ABB RobotStudio station: IRB120 Writing.rsstn

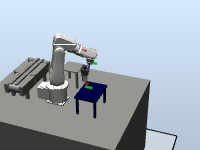
Station Solution4 (saved by RobotStudio 6.8.8148.134)
Controller System1, task T_ROB1: task frame (RAPID world) sits at (85.62, 36.2, 947.96) mm, rotated rx 0 ry 0 rz 180 deg in the station
Controller System1
  mechanical unit ROB_1: IRB120_3_58__01, 6 joints, base frame (0, 0, 0) mm
Layout (positions relative to the parent item):
  - 零件1 [part] at (0, 0, 512.15) mm, rotated rx 90 ry 0 rz 0 deg
  - 写字台 [part] at (-381.08, 197.71, 1142.77) mm, rotated rx 90 ry 0 rz 0 deg
  - 字 [part] at (-241.46, 516.73, 1142.95) mm, rotated rx 90 ry 0 rz 90 deg
  - IRB120_3_58__01 [mechanism, from Robots\IRB120_3_58_G_01.rslib] at (85.62, 36.2, 947.96) mm, rotated rx 0 ry 0 rz 180 deg; joint values [0.5258, 0.1426, 0.3629, -0.5655, 1.4593, 2.276] (rad or m)
  - MyTool [mechanism, from Training Objects\myTool.rslib] at (-205.42, -88.36, 1363.49) mm, rotated rx -180 ry 38 rz -90 deg
  - SmartComponent_1 [smart component]
      signals: DI diTCP
      connections:
        SmartComponent_1.diTCP -> TraceTCP.Enabled
    - TraceTCP [smart component, from Components\TraceTCP.rslib]
        properties: Robot=IRB120_3_58__01
Attachment: MyTool is attached to IRB120_3_58__01 / Link6
Station logic (signal -> signal, property => property):
  System1.doTCP0 -> SmartComponent_1.diTCP
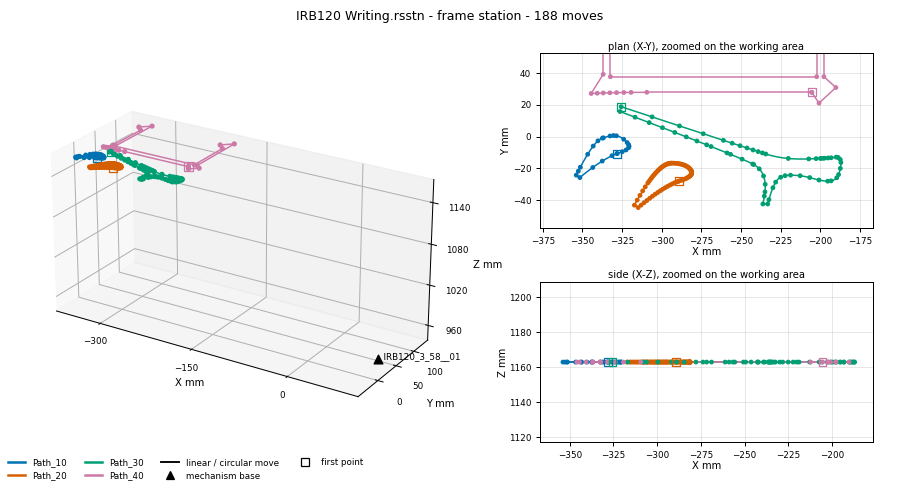
[picture p0: tool path of IRB120 Writing.rsstn in frame station, 188 of 188 moves have a stored position in this frame; points joined in program order, loops and branches not executed]
Targets, tools, work objects and paths stored in the station, written as RAPID:
! task T_ROB1
MODULE Module1
  PERS tooldata MyTool:=[TRUE,[[31.792631019,0,229.638935148],[0.945518576,0,0.325568154,0]],[1,[0,0,1],[1,0,0,0],0,0,0]];
  CONST robtarget Target_10:=[[413.794181769,46.847111716,214.996798109],[0,-0.157825043,0.987467091,0],[0,0,0,0],[9E+09,9E+09,9E+09,9E+09,9E+09,9E+09]];
  CONST robtarget Target_20:=[[415.060758139,47.36953404,214.996798109],[0,-0.157825043,0.987467091,0],[0,0,0,0],[9E+09,9E+09,9E+09,9E+09,9E+09,9E+09]];
  CONST robtarget Target_30:=[[416.985055299,48.218994242,214.996798109],[0,-0.157825043,0.987467091,0],[0,0,0,0],[9E+09,9E+09,9E+09,9E+09,9E+09,9E+09]];
  CONST robtarget Target_40:=[[420.337020954,49.9590146,214.996798109],[0,-0.157825043,0.987467091,0],[0,0,0,0],[9E+09,9E+09,9E+09,9E+09,9E+09,9E+09]];
  CONST robtarget Target_50:=[[423.156723452,51.613418661,214.996798109],[0,-0.157825043,0.987467091,0],[0,0,0,0],[9E+09,9E+09,9E+09,9E+09,9E+09,9E+09]];
  CONST robtarget Target_60:=[[426.087811207,53.506801611,214.996798109],[0,-0.157825043,0.987467091,0],[0,0,0,0],[9E+09,9E+09,9E+09,9E+09,9E+09,9E+09]];
  CONST robtarget Target_70:=[[429.127715578,55.643607322,214.996798109],[0,-0.157825043,0.987467091,0],[0,0,0,0],[9E+09,9E+09,9E+09,9E+09,9E+09,9E+09]];
  CONST robtarget Target_80:=[[433.930399717,59.270989922,214.996798109],[0,-0.157825043,0.987467091,0],[0,0,0,0],[9E+09,9E+09,9E+09,9E+09,9E+09,9E+09]];
  CONST robtarget Target_90:=[[437.267739461,61.991342486,214.996798109],[0,-0.157825043,0.987467091,0],[0,0,0,0],[9E+09,9E+09,9E+09,9E+09,9E+09,9E+09]];
  CONST robtarget Target_100:=[[439.539374076,60.476919409,214.996798109],[0,-0.157825043,0.987467091,0],[0,0,0,0],[9E+09,9E+09,9E+09,9E+09,9E+09,9E+09]];
  CONST robtarget Target_110:=[[438.254894214,57.978091262,214.996798109],[0,-0.157825043,0.987467091,0],[0,0,0,0],[9E+09,9E+09,9E+09,9E+09,9E+09,9E+09]];
  CONST robtarget Target_120:=[[436.959245871,55.484932229,214.996798109],[0,-0.157825043,0.987467091,0],[0,0,0,0],[9E+09,9E+09,9E+09,9E+09,9E+09,9E+09]];
  CONST robtarget Target_130:=[[434.575431769,51.081887357,214.996798109],[0,-0.157825043,0.987467091,0],[0,0,0,0],[9E+09,9E+09,9E+09,9E+09,9E+09,9E+09]];
  CONST robtarget Target_140:=[[432.331842025,47.295829665,214.996798109],[0,-0.157825043,0.987467091,0],[0,0,0,0],[9E+09,9E+09,9E+09,9E+09,9E+09,9E+09]];
  CONST robtarget Target_150:=[[430.790454976,44.888264366,214.996798109],[0,-0.157825043,0.987467091,0],[0,0,0,0],[9E+09,9E+09,9E+09,9E+09,9E+09,9E+09]];
  CONST robtarget Target_160:=[[428.845408894,42.148797629,214.996798109],[0,-0.157825043,0.987467091,0],[0,0,0,0],[9E+09,9E+09,9E+09,9E+09,9E+09,9E+09]];
  CONST robtarget Target_170:=[[427.504490728,40.516553609,214.996798109],[0,-0.157825043,0.987467091,0],[0,0,0,0],[9E+09,9E+09,9E+09,9E+09,9E+09,9E+09]];
  CONST robtarget Target_180:=[[425.856041428,38.831157314,214.996798109],[0,-0.157825043,0.987467091,0],[0,0,0,0],[9E+09,9E+09,9E+09,9E+09,9E+09,9E+09]];
  CONST robtarget Target_190:=[[424.358135134,37.755273557,214.996798109],[0,-0.157825043,0.987467091,0],[0,0,0,0],[9E+09,9E+09,9E+09,9E+09,9E+09,9E+09]];
  CONST robtarget Target_200:=[[423.034428232,37.149604926,214.996798109],[0,-0.157825043,0.987467091,0],[0,0,0,0],[9E+09,9E+09,9E+09,9E+09,9E+09,9E+09]];
  CONST robtarget Target_210:=[[422.419010763,36.934235315,214.996798109],[0,-0.157825043,0.987467091,0],[0,0,0,0],[9E+09,9E+09,9E+09,9E+09,9E+09,9E+09]];
  CONST robtarget Target_220:=[[420.134296252,36.25336216,214.996798109],[0,-0.157825043,0.987467091,0],[0,0,0,0],[9E+09,9E+09,9E+09,9E+09,9E+09,9E+09]];
  CONST robtarget Target_230:=[[418.244052483,35.756988405,214.996798109],[0,-0.157825043,0.987467091,0],[0,0,0,0],[9E+09,9E+09,9E+09,9E+09,9E+09,9E+09]];
  CONST robtarget Target_240:=[[417.383925358,35.601118127,214.996798109],[0,-0.157825043,0.987467091,0],[0,0,0,0],[9E+09,9E+09,9E+09,9E+09,9E+09,9E+09]];
  CONST robtarget Target_250:=[[416.065816384,35.48893864,214.996798109],[0,-0.157825043,0.987467091,0],[0,0,0,0],[9E+09,9E+09,9E+09,9E+09,9E+09,9E+09]];
  CONST robtarget Target_260:=[[415.135685534,35.543807614,214.996798109],[0,-0.157825043,0.987467091,0],[0,0,0,0],[9E+09,9E+09,9E+09,9E+09,9E+09,9E+09]];
  CONST robtarget Target_270:=[[414.214854846,35.65720787,214.996798109],[0,-0.157825043,0.987467091,0],[0,0,0,0],[9E+09,9E+09,9E+09,9E+09,9E+09,9E+09]];
  CONST robtarget Target_280:=[[411.628963846,36.531651758,214.996798109],[0,-0.157825043,0.987467091,0],[0,0,0,0],[9E+09,9E+09,9E+09,9E+09,9E+09,9E+09]];
  CONST robtarget Target_290:=[[409.628567412,37.837626066,214.996798109],[0,-0.157825043,0.987467091,0],[0,0,0,0],[9E+09,9E+09,9E+09,9E+09,9E+09,9E+09]];
  CONST robtarget Target_300:=[[408.575369643,38.75449417,214.996798109],[0,-0.157825043,0.987467091,0],[0,0,0,0],[9E+09,9E+09,9E+09,9E+09,9E+09,9E+09]];
  CONST robtarget Target_310:=[[407.440478174,39.932033456,214.996798109],[0,-0.157825043,0.987467091,0],[0,0,0,0],[9E+09,9E+09,9E+09,9E+09,9E+09,9E+09]];
  CONST robtarget Target_320:=[[406.979277923,40.508970691,214.996798109],[0,-0.157825043,0.987467091,0],[0,0,0,0],[9E+09,9E+09,9E+09,9E+09,9E+09,9E+09]];
  CONST robtarget Target_330:=[[406.528343034,41.21067125,214.996798109],[0,-0.157825043,0.987467091,0],[0,0,0,0],[9E+09,9E+09,9E+09,9E+09,9E+09,9E+09]];
  CONST robtarget Target_340:=[[406.352602418,41.666682817,214.996798109],[0,-0.157825043,0.987467091,0],[0,0,0,0],[9E+09,9E+09,9E+09,9E+09,9E+09,9E+09]];
  CONST robtarget Target_350:=[[406.222066384,42.303842486,214.996798109],[0,-0.157825043,0.987467091,0],[0,0,0,0],[9E+09,9E+09,9E+09,9E+09,9E+09,9E+09]];
  CONST robtarget Target_360:=[[406.291553057,42.730004792,214.996798109],[0,-0.157825043,0.987467091,0],[0,0,0,0],[9E+09,9E+09,9E+09,9E+09,9E+09,9E+09]];
  CONST robtarget Target_370:=[[406.491071898,43.157591418,214.996798109],[0,-0.157825043,0.987467091,0],[0,0,0,0],[9E+09,9E+09,9E+09,9E+09,9E+09,9E+09]];
  CONST robtarget Target_380:=[[407.287771512,44.014579665,214.996798109],[0,-0.157825043,0.987467091,0],[0,0,0,0],[9E+09,9E+09,9E+09,9E+09,9E+09,9E+09]];
  CONST robtarget Target_390:=[[408.129117666,44.575477101,214.996798109],[0,-0.157825043,0.987467091,0],[0,0,0,0],[9E+09,9E+09,9E+09,9E+09,9E+09,9E+09]];
  CONST robtarget Target_400:=[[409.166777923,45.136374537,214.996798109],[0,-0.157825043,0.987467091,0],[0,0,0,0],[9E+09,9E+09,9E+09,9E+09,9E+09,9E+09]];
  CONST robtarget Target_410:=[[410.484886897,45.697271973,214.996798109],[0,-0.157825043,0.987467091,0],[0,0,0,0],[9E+09,9E+09,9E+09,9E+09,9E+09,9E+09]];
  CONST robtarget Target_420:=[[412.027354846,46.286214281,214.996798109],[0,-0.157825043,0.987467091,0],[0,0,0,0],[9E+09,9E+09,9E+09,9E+09,9E+09,9E+09]];
  CONST robtarget Target_430:=[[413.794181769,46.847111716,214.996798109],[0,-0.157825043,0.987467091,0],[0,0,0,0],[9E+09,9E+09,9E+09,9E+09,9E+09,9E+09]];
  CONST robtarget Target_440:=[[375.008124076,64.262977101,214.996798109],[0,0.417358337,0.908741998,0],[0,0,0,0],[9E+09,9E+09,9E+09,9E+09,9E+09,9E+09]];
  CONST robtarget Target_450:=[[376.346419308,64.795791588,214.996798109],[0,0.417358337,0.908741998,0],[0,0,0,0],[9E+09,9E+09,9E+09,9E+09,9E+09,9E+09]];
  CONST robtarget Target_460:=[[377.672386897,65.356727101,214.996798109],[0,0.417358337,0.908741998,0],[0,0,0,0],[9E+09,9E+09,9E+09,9E+09,9E+09,9E+09]];
  CONST robtarget Target_470:=[[379.085741747,66.020298008,214.996798109],[0,0.417358337,0.908741998,0],[0,0,0,0],[9E+09,9E+09,9E+09,9E+09,9E+09,9E+09]];
  CONST robtarget Target_480:=[[380.476874076,66.730925819,214.996798109],[0,0.417358337,0.908741998,0],[0,0,0,0],[9E+09,9E+09,9E+09,9E+09,9E+09,9E+09]];
  CONST robtarget Target_490:=[[381.973257971,67.540696014,214.996798109],[0,0.417358337,0.908741998,0],[0,0,0,0],[9E+09,9E+09,9E+09,9E+09,9E+09,9E+09]];
  CONST robtarget Target_500:=[[383.449630487,68.385573255,214.996798109],[0,0.417358337,0.908741998,0],[0,0,0,0],[9E+09,9E+09,9E+09,9E+09,9E+09,9E+09]];
  CONST robtarget Target_510:=[[385.016861186,69.33557153,214.996798109],[0,0.417358337,0.908741998,0],[0,0,0,0],[9E+09,9E+09,9E+09,9E+09,9E+09,9E+09]];
  CONST robtarget Target_520:=[[386.562611256,70.320669409,214.996798109],[0,0.417358337,0.908741998,0],[0,0,0,0],[9E+09,9E+09,9E+09,9E+09,9E+09,9E+09]];
  CONST robtarget Target_530:=[[388.201363528,71.410852065,214.996798109],[0,0.417358337,0.908741998,0],[0,0,0,0],[9E+09,9E+09,9E+09,9E+09,9E+09,9E+09]];
  CONST robtarget Target_540:=[[389.815816384,72.536214281,214.996798109],[0,0.417358337,0.908741998,0],[0,0,0,0],[9E+09,9E+09,9E+09,9E+09,9E+09,9E+09]];
  CONST robtarget Target_550:=[[391.522124522,73.785045315,214.996798109],[0,0.417358337,0.908741998,0],[0,0,0,0],[9E+09,9E+09,9E+09,9E+09,9E+09,9E+09]];
  CONST robtarget Target_560:=[[393.209245871,75.060252742,214.996798109],[0,0.417358337,0.908741998,0],[0,0,0,0],[9E+09,9E+09,9E+09,9E+09,9E+09,9E+09]];
  CONST robtarget Target_570:=[[394.999763377,76.436392584,214.996798109],[0,0.417358337,0.908741998,0],[0,0,0,0],[9E+09,9E+09,9E+09,9E+09,9E+09,9E+09]];
  CONST robtarget Target_580:=[[396.770944589,77.83669505,214.996798109],[0,0.417358337,0.908741998,0],[0,0,0,0],[9E+09,9E+09,9E+09,9E+09,9E+09,9E+09]];
  CONST robtarget Target_590:=[[398.630982599,79.367934635,214.996798109],[0,0.417358337,0.908741998,0],[0,0,0,0],[9E+09,9E+09,9E+09,9E+09,9E+09,9E+09]];
  CONST robtarget Target_600:=[[400.472867666,80.921630947,214.996798109],[0,0.417358337,0.908741998,0],[0,0,0,0],[9E+09,9E+09,9E+09,9E+09,9E+09,9E+09]];
  CONST robtarget Target_610:=[[402.856681769,79.40720787,214.996798109],[0,0.417358337,0.908741998,0],[0,0,0,0],[9E+09,9E+09,9E+09,9E+09,9E+09,9E+09]];
  CONST robtarget Target_620:=[[401.089854846,76.210092486,214.996798109],[0,0.417358337,0.908741998,0],[0,0,0,0],[9E+09,9E+09,9E+09,9E+09,9E+09,9E+09]];
  CONST robtarget Target_630:=[[399.351072794,73.209291204,214.996798109],[0,0.417358337,0.908741998,0],[0,0,0,0],[9E+09,9E+09,9E+09,9E+09,9E+09,9E+09]];
  CONST robtarget Target_640:=[[397.668380487,70.404804024,214.996798109],[0,0.417358337,0.908741998,0],[0,0,0,0],[9E+09,9E+09,9E+09,9E+09,9E+09,9E+09]];
  CONST robtarget Target_650:=[[396.013733051,67.824675819,214.996798109],[0,0.417358337,0.908741998,0],[0,0,0,0],[9E+09,9E+09,9E+09,9E+09,9E+09,9E+09]];
  CONST robtarget Target_660:=[[394.415175358,65.440861716,214.996798109],[0,0.417358337,0.908741998,0],[0,0,0,0],[9E+09,9E+09,9E+09,9E+09,9E+09,9E+09]];
  CONST robtarget Target_670:=[[393.639289698,64.340440715,214.996798109],[0,0.417358337,0.908741998,0],[0,0,0,0],[9E+09,9E+09,9E+09,9E+09,9E+09,9E+09]];
  CONST robtarget Target_680:=[[392.844662538,63.253361716,214.996798109],[0,0.417358337,0.908741998,0],[0,0,0,0],[9E+09,9E+09,9E+09,9E+09,9E+09,9E+09]];
  CONST robtarget Target_690:=[[392.096719617,62.264585202,214.996798109],[0,0.417358337,0.908741998,0],[0,0,0,0],[9E+09,9E+09,9E+09,9E+09,9E+09,9E+09]];
  CONST robtarget Target_700:=[[391.330239461,61.290220691,214.996798109],[0,0.417358337,0.908741998,0],[0,0,0,0],[9E+09,9E+09,9E+09,9E+09,9E+09,9E+09]];
  CONST robtarget Target_710:=[[390.596978307,60.39852615,214.996798109],[0,0.417358337,0.908741998,0],[0,0,0,0],[9E+09,9E+09,9E+09,9E+09,9E+09,9E+09]];
  CONST robtarget Target_720:=[[389.843861256,59.523393768,214.996798109],[0,0.417358337,0.908741998,0],[0,0,0,0],[9E+09,9E+09,9E+09,9E+09,9E+09,9E+09]];
  CONST robtarget Target_730:=[[389.139301128,58.742195279,214.996798109],[0,0.417358337,0.908741998,0],[0,0,0,0],[9E+09,9E+09,9E+09,9E+09,9E+09,9E+09]];
  CONST robtarget Target_740:=[[388.413572794,57.980925819,214.996798109],[0,0.417358337,0.908741998,0],[0,0,0,0],[9E+09,9E+09,9E+09,9E+09,9E+09,9E+09]];
  CONST robtarget Target_750:=[[387.721616611,57.298552386,214.996798109],[0,0.417358337,0.908741998,0],[0,0,0,0],[9E+09,9E+09,9E+09,9E+09,9E+09,9E+09]];
  CONST robtarget Target_760:=[[387.011329205,56.634771973,214.996798109],[0,0.417358337,0.908741998,0],[0,0,0,0],[9E+09,9E+09,9E+09,9E+09,9E+09,9E+09]];
  CONST robtarget Target_770:=[[386.349253035,56.04656752,214.996798109],[0,0.417358337,0.908741998,0],[0,0,0,0],[9E+09,9E+09,9E+09,9E+09,9E+09,9E+09]];
  CONST robtarget Target_780:=[[385.665175358,55.484932229,214.996798109],[0,0.417358337,0.908741998,0],[0,0,0,0],[9E+09,9E+09,9E+09,9E+09,9E+09,9E+09]];
  CONST robtarget Target_790:=[[385.017465851,55.006494103,214.996798109],[0,0.417358337,0.908741998,0],[0,0,0,0],[9E+09,9E+09,9E+09,9E+09,9E+09,9E+09]];
  CONST robtarget Target_800:=[[384.347066384,54.55945146,214.996798109],[0,0.417358337,0.908741998,0],[0,0,0,0],[9E+09,9E+09,9E+09,9E+09,9E+09,9E+09]];
  CONST robtarget Target_810:=[[383.712063268,54.176492085,214.996798109],[0,0.417358337,0.908741998,0],[0,0,0,0],[9E+09,9E+09,9E+09,9E+09,9E+09,9E+09]];
  CONST robtarget Target_820:=[[383.057002281,53.830284793,214.996798109],[0,0.417358337,0.908741998,0],[0,0,0,0],[9E+09,9E+09,9E+09,9E+09,9E+09,9E+09]];
  CONST robtarget Target_830:=[[382.448312966,53.558411366,214.996798109],[0,0.417358337,0.908741998,0],[0,0,0,0],[9E+09,9E+09,9E+09,9E+09,9E+09,9E+09]];
  CONST robtarget Target_840:=[[381.823027923,53.325477101,214.996798109],[0,0.417358337,0.908741998,0],[0,0,0,0],[9E+09,9E+09,9E+09,9E+09,9E+09,9E+09]];
  CONST robtarget Target_850:=[[381.239521236,53.148696158,214.996798109],[0,0.417358337,0.908741998,0],[0,0,0,0],[9E+09,9E+09,9E+09,9E+09,9E+09,9E+09]];
  CONST robtarget Target_860:=[[380.645143307,53.016983511,214.996798109],[0,0.417358337,0.908741998,0],[0,0,0,0],[9E+09,9E+09,9E+09,9E+09,9E+09,9E+09]];
  CONST robtarget Target_870:=[[380.072473159,52.941341422,214.996798109],[0,0.417358337,0.908741998,0],[0,0,0,0],[9E+09,9E+09,9E+09,9E+09,9E+09,9E+09]];
  CONST robtarget Target_880:=[[379.495303564,52.904804024,214.996798109],[0,0.417358337,0.908741998,0],[0,0,0,0],[9E+09,9E+09,9E+09,9E+09,9E+09,9E+09]];
  CONST robtarget Target_890:=[[378.415082007,52.904711962,214.996798109],[0,0.417358337,0.908741998,0],[0,0,0,0],[9E+09,9E+09,9E+09,9E+09,9E+09,9E+09]];
  CONST robtarget Target_900:=[[377.335848435,52.960893768,214.996798109],[0,0.417358337,0.908741998,0],[0,0,0,0],[9E+09,9E+09,9E+09,9E+09,9E+09,9E+09]];
  CONST robtarget Target_910:=[[376.338043667,53.040496731,214.996798109],[0,0.417358337,0.908741998,0],[0,0,0,0],[9E+09,9E+09,9E+09,9E+09,9E+09,9E+09]];
  CONST robtarget Target_920:=[[375.344662538,53.15720787,214.996798109],[0,0.417358337,0.908741998,0],[0,0,0,0],[9E+09,9E+09,9E+09,9E+09,9E+09,9E+09]];
  CONST robtarget Target_930:=[[374.457782164,53.305987403,214.996798109],[0,0.417358337,0.908741998,0],[0,0,0,0],[9E+09,9E+09,9E+09,9E+09,9E+09,9E+09]];
  CONST robtarget Target_940:=[[373.577835615,53.493746332,214.996798109],[0,0.417358337,0.908741998,0],[0,0,0,0],[9E+09,9E+09,9E+09,9E+09,9E+09,9E+09]];
  CONST robtarget Target_950:=[[372.773048016,53.698879505,214.996798109],[0,0.417358337,0.908741998,0],[0,0,0,0],[9E+09,9E+09,9E+09,9E+09,9E+09,9E+09]];
  CONST robtarget Target_960:=[[371.979277923,53.942464281,214.996798109],[0,0.417358337,0.908741998,0],[0,0,0,0],[9E+09,9E+09,9E+09,9E+09,9E+09,9E+09]];
  CONST robtarget Target_970:=[[371.254081393,54.212783325,214.996798109],[0,0.417358337,0.908741998,0],[0,0,0,0],[9E+09,9E+09,9E+09,9E+09,9E+09,9E+09]];
  CONST robtarget Target_980:=[[370.548989461,54.531406588,214.996798109],[0,0.417358337,0.908741998,0],[0,0,0,0],[9E+09,9E+09,9E+09,9E+09,9E+09,9E+09]];
  CONST robtarget Target_990:=[[369.919037638,54.873733121,214.996798109],[0,0.417358337,0.908741998,0],[0,0,0,0],[9E+09,9E+09,9E+09,9E+09,9E+09,9E+09]];
  CONST robtarget Target_1000:=[[369.315015102,55.260573255,214.996798109],[0,0.417358337,0.908741998,0],[0,0,0,0],[9E+09,9E+09,9E+09,9E+09,9E+09,9E+09]];
  CONST robtarget Target_1010:=[[368.779066824,55.660499694,214.996798109],[0,0.417358337,0.908741998,0],[0,0,0,0],[9E+09,9E+09,9E+09,9E+09,9E+09,9E+09]];
  CONST robtarget Target_1020:=[[368.277354846,56.101919409,214.996798109],[0,0.417358337,0.908741998,0],[0,0,0,0],[9E+09,9E+09,9E+09,9E+09,9E+09,9E+09]];
  CONST robtarget Target_1030:=[[367.832868118,56.571926989,214.996798109],[0,0.417358337,0.908741998,0],[0,0,0,0],[9E+09,9E+09,9E+09,9E+09,9E+09,9E+09]];
  CONST robtarget Target_1040:=[[367.436008692,57.083489922,214.996798109],[0,0.417358337,0.908741998,0],[0,0,0,0],[9E+09,9E+09,9E+09,9E+09,9E+09,9E+09]];
  CONST robtarget Target_1050:=[[367.134505638,57.569713902,214.996798109],[0,0.417358337,0.908741998,0],[0,0,0,0],[9E+09,9E+09,9E+09,9E+09,9E+09,9E+09]];
  CONST robtarget Target_1060:=[[367.008335929,57.826391072,214.996798109],[0,0.417358337,0.908741998,0],[0,0,0,0],[9E+09,9E+09,9E+09,9E+09,9E+09,9E+09]];
  CONST robtarget Target_1070:=[[366.903156128,58.093105306,214.996798109],[0,0.417358337,0.908741998,0],[0,0,0,0],[9E+09,9E+09,9E+09,9E+09,9E+09,9E+09]];
  CONST robtarget Target_1080:=[[366.831717767,58.332956921,214.996798109],[0,0.417358337,0.908741998,0],[0,0,0,0],[9E+09,9E+09,9E+09,9E+09,9E+09,9E+09]];
  CONST robtarget Target_1090:=[[366.782207519,58.578278493,214.996798109],[0,0.417358337,0.908741998,0],[0,0,0,0],[9E+09,9E+09,9E+09,9E+09,9E+09,9E+09]];
  CONST robtarget Target_1100:=[[366.758115486,58.8264061,214.996798109],[0,0.417358337,0.908741998,0],[0,0,0,0],[9E+09,9E+09,9E+09,9E+09,9E+09,9E+09]];
  CONST robtarget Target_1110:=[[366.762931769,59.074675819,214.996798109],[0,0.417358337,0.908741998,0],[0,0,0,0],[9E+09,9E+09,9E+09,9E+09,9E+09,9E+09]];
  CONST robtarget Target_1120:=[[366.799526296,59.323087626,214.996798109],[0,0.417358337,0.908741998,0],[0,0,0,0],[9E+09,9E+09,9E+09,9E+09,9E+09,9E+09]];
  CONST robtarget Target_1130:=[[366.86557166,59.566456761,214.996798109],[0,0.417358337,0.908741998,0],[0,0,0,0],[9E+09,9E+09,9E+09,9E+09,9E+09,9E+09]];
  CONST robtarget Target_1140:=[[366.957420476,59.802316835,214.996798109],[0,0.417358337,0.908741998,0],[0,0,0,0],[9E+09,9E+09,9E+09,9E+09,9E+09,9E+09]];
  CONST robtarget Target_1150:=[[367.071425358,60.02820146,214.996798109],[0,0.417358337,0.908741998,0],[0,0,0,0],[9E+09,9E+09,9E+09,9E+09,9E+09,9E+09]];
  CONST robtarget Target_1160:=[[367.231695097,60.282194269,214.996798109],[0,0.417358337,0.908741998,0],[0,0,0,0],[9E+09,9E+09,9E+09,9E+09,9E+09,9E+09]];
  CONST robtarget Target_1170:=[[367.414118042,60.520052905,214.996798109],[0,0.417358337,0.908741998,0],[0,0,0,0],[9E+09,9E+09,9E+09,9E+09,9E+09,9E+09]];
  CONST robtarget Target_1180:=[[367.828636897,60.953682229,214.996798109],[0,0.417358337,0.908741998,0],[0,0,0,0],[9E+09,9E+09,9E+09,9E+09,9E+09,9E+09]];
  CONST robtarget Target_1190:=[[368.383395251,61.415334756,214.996798109],[0,0.417358337,0.908741998,0],[0,0,0,0],[9E+09,9E+09,9E+09,9E+09,9E+09,9E+09]];
  CONST robtarget Target_1200:=[[368.97847664,61.823073255,214.996798109],[0,0.417358337,0.908741998,0],[0,0,0,0],[9E+09,9E+09,9E+09,9E+09,9E+09,9E+09]];
  CONST robtarget Target_1210:=[[369.749959866,62.269156545,214.996798109],[0,0.417358337,0.908741998,0],[0,0,0,0],[9E+09,9E+09,9E+09,9E+09,9E+09,9E+09]];
  CONST robtarget Target_1220:=[[370.548989461,62.664419409,214.996798109],[0,0.417358337,0.908741998,0],[0,0,0,0],[9E+09,9E+09,9E+09,9E+09,9E+09,9E+09]];
  CONST robtarget Target_1230:=[[371.549209209,63.094640164,214.996798109],[0,0.417358337,0.908741998,0],[0,0,0,0],[9E+09,9E+09,9E+09,9E+09,9E+09,9E+09]];
  CONST robtarget Target_1240:=[[372.56822023,63.477720691,214.996798109],[0,0.417358337,0.908741998,0],[0,0,0,0],[9E+09,9E+09,9E+09,9E+09,9E+09,9E+09]];
  CONST robtarget Target_1250:=[[373.783847633,63.883294038,214.996798109],[0,0.417358337,0.908741998,0],[0,0,0,0],[9E+09,9E+09,9E+09,9E+09,9E+09,9E+09]];
  CONST robtarget Target_1260:=[[375.008124076,64.262977101,214.996798109],[0,0.417358337,0.908741998,0],[0,0,0,0],[9E+09,9E+09,9E+09,9E+09,9E+09,9E+09]];
  CONST robtarget Target_1270:=[[411.186008692,17.315861716,214.996798109],[0,0.150905267,0.988548229,0],[0,0,0,0],[9E+09,9E+09,9E+09,9E+09,9E+09,9E+09]];
  CONST robtarget Target_1280:=[[391.694822794,23.738137357,214.996798109],[0,0.150905267,0.988548229,0],[0,0,0,0],[9E+09,9E+09,9E+09,9E+09,9E+09,9E+09]];
  CONST robtarget Target_1290:=[[374.44722664,29.431246332,214.996798109],[0,0.150905267,0.988548229,0],[0,0,0,0],[9E+09,9E+09,9E+09,9E+09,9E+09,9E+09]];
  CONST robtarget Target_1300:=[[359.44322023,34.339098896,214.996798109],[0,0.150905267,0.988548229,0],[0,0,0,0],[9E+09,9E+09,9E+09,9E+09,9E+09,9E+09]];
  CONST robtarget Target_1310:=[[346.738893307,38.517784793,214.996798109],[0,0.150905267,0.988548229,0],[0,0,0,0],[9E+09,9E+09,9E+09,9E+09,9E+09,9E+09]];
  CONST robtarget Target_1320:=[[341.214053564,40.312656588,214.996798109],[0,0.150905267,0.988548229,0],[0,0,0,0],[9E+09,9E+09,9E+09,9E+09,9E+09,9E+09]];
  CONST robtarget Target_1330:=[[336.250111256,41.911214281,214.996798109],[0,0.150905267,0.988548229,0],[0,0,0,0],[9E+09,9E+09,9E+09,9E+09,9E+09,9E+09]];
  CONST robtarget Target_1340:=[[331.875111256,43.341502742,214.996798109],[0,0.150905267,0.988548229,0],[0,0,0,0],[9E+09,9E+09,9E+09,9E+09,9E+09,9E+09]];
  CONST robtarget Target_1350:=[[328.061008692,44.575477101,214.996798109],[0,0.150905267,0.988548229,0],[0,0,0,0],[9E+09,9E+09,9E+09,9E+09,9E+09,9E+09]];
  CONST robtarget Target_1360:=[[324.807803564,45.613137357,214.996798109],[0,0.150905267,0.988548229,0],[0,0,0,0],[9E+09,9E+09,9E+09,9E+09,9E+09,9E+09]];
  CONST robtarget Target_1370:=[[322.115495871,46.454483511,214.996798109],[0,0.150905267,0.988548229,0],[0,0,0,0],[9E+09,9E+09,9E+09,9E+09,9E+09,9E+09]];
  CONST robtarget Target_1380:=[[319.984085615,47.127560434,214.996798109],[0,0.150905267,0.988548229,0],[0,0,0,0],[9E+09,9E+09,9E+09,9E+09,9E+09,9E+09]];
  CONST robtarget Target_1390:=[[313.085047153,48.894387357,214.996798109],[0,0.150905267,0.988548229,0],[0,0,0,0],[9E+09,9E+09,9E+09,9E+09,9E+09,9E+09]];
  CONST robtarget Target_1400:=[[305.818359796,49.950656798,214.996798109],[0,0.150905267,0.988548229,0],[0,0,0,0],[9E+09,9E+09,9E+09,9E+09,9E+09,9E+09]];
  CONST robtarget Target_1410:=[[299.518531514,50.285951425,214.996798109],[0,0.150905267,0.988548229,0],[0,0,0,0],[9E+09,9E+09,9E+09,9E+09,9E+09,9E+09]];
  CONST robtarget Target_1420:=[[292.934639214,50.217640377,214.996798109],[0,0.150905267,0.988548229,0],[0,0,0,0],[9E+09,9E+09,9E+09,9E+09,9E+09,9E+09]];
  CONST robtarget Target_1430:=[[288.293380487,50.044227101,214.996798109],[0,0.150905267,0.988548229,0],[0,0,0,0],[9E+09,9E+09,9E+09,9E+09,9E+09,9E+09]];
  CONST robtarget Target_1440:=[[285.516938179,49.932047614,214.996798109],[0,0.150905267,0.988548229,0],[0,0,0,0],[9E+09,9E+09,9E+09,9E+09,9E+09,9E+09]];
  CONST robtarget Target_1450:=[[284.26848519,49.869507835,214.996798109],[0,0.150905267,0.988548229,0],[0,0,0,0],[9E+09,9E+09,9E+09,9E+09,9E+09,9E+09]];
  CONST robtarget Target_1460:=[[283.020944589,49.791823255,214.996798109],[0,0.150905267,0.988548229,0],[0,0,0,0],[9E+09,9E+09,9E+09,9E+09,9E+09,9E+09]];
  CONST robtarget Target_1470:=[[280.805399717,49.623554024,214.996798109],[0,0.150905267,0.988548229,0],[0,0,0,0],[9E+09,9E+09,9E+09,9E+09,9E+09,9E+09]];
  CONST robtarget Target_1480:=[[278.81421382,49.483329665,214.996798109],[0,0.150905267,0.988548229,0],[0,0,0,0],[9E+09,9E+09,9E+09,9E+09,9E+09,9E+09]];
  CONST robtarget Target_1490:=[[277.10347664,49.315060434,214.996798109],[0,0.150905267,0.988548229,0],[0,0,0,0],[9E+09,9E+09,9E+09,9E+09,9E+09,9E+09]];
  CONST robtarget Target_1500:=[[275.645143307,49.118746332,214.996798109],[0,0.150905267,0.988548229,0],[0,0,0,0],[9E+09,9E+09,9E+09,9E+09,9E+09,9E+09]];
  CONST robtarget Target_1510:=[[274.969747093,49.178976609,214.996798109],[0,0.150905267,0.988548229,0],[0,0,0,0],[9E+09,9E+09,9E+09,9E+09,9E+09,9E+09]];
  CONST robtarget Target_1520:=[[274.327034333,49.343105306,214.996798109],[0,0.150905267,0.988548229,0],[0,0,0,0],[9E+09,9E+09,9E+09,9E+09,9E+09,9E+09]];
  CONST robtarget Target_1530:=[[273.576969861,49.845534873,214.996798109],[0,0.150905267,0.988548229,0],[0,0,0,0],[9E+09,9E+09,9E+09,9E+09,9E+09,9E+09]];
  CONST robtarget Target_1540:=[[273.031415049,50.632272341,214.996798109],[0,0.150905267,0.988548229,0],[0,0,0,0],[9E+09,9E+09,9E+09,9E+09,9E+09,9E+09]];
  CONST robtarget Target_1550:=[[272.726969299,51.657724944,214.996798109],[0,0.150905267,0.988548229,0],[0,0,0,0],[9E+09,9E+09,9E+09,9E+09,9E+09,9E+09]];
  CONST robtarget Target_1560:=[[272.639258943,52.486789663,214.996798109],[0,0.150905267,0.988548229,0],[0,0,0,0],[9E+09,9E+09,9E+09,9E+09,9E+09,9E+09]];
  CONST robtarget Target_1570:=[[272.700431769,54.503361716,214.996798109],[0,0.150905267,0.988548229,0],[0,0,0,0],[9E+09,9E+09,9E+09,9E+09,9E+09,9E+09]];
  CONST robtarget Target_1580:=[[273.008925358,56.214098896,214.996798109],[0,0.150905267,0.988548229,0],[0,0,0,0],[9E+09,9E+09,9E+09,9E+09,9E+09,9E+09]];
  CONST robtarget Target_1590:=[[273.457643307,58.093105306,214.996798109],[0,0.150905267,0.988548229,0],[0,0,0,0],[9E+09,9E+09,9E+09,9E+09,9E+09,9E+09]];
  CONST robtarget Target_1600:=[[274.13072023,60.112336075,214.996798109],[0,0.150905267,0.988548229,0],[0,0,0,0],[9E+09,9E+09,9E+09,9E+09,9E+09,9E+09]];
  CONST robtarget Target_1610:=[[274.559010932,61.062267847,214.996798109],[0,0.150905267,0.988548229,0],[0,0,0,0],[9E+09,9E+09,9E+09,9E+09,9E+09,9E+09]];
  CONST robtarget Target_1620:=[[275.268769542,62.12463988,214.996798109],[0,0.150905267,0.988548229,0],[0,0,0,0],[9E+09,9E+09,9E+09,9E+09,9E+09,9E+09]];
  CONST robtarget Target_1630:=[[276.826598747,63.357179665,214.996798109],[0,0.150905267,0.988548229,0],[0,0,0,0],[9E+09,9E+09,9E+09,9E+09,9E+09,9E+09]];
  CONST robtarget Target_1640:=[[278.829760733,64.072101822,214.996798109],[0,0.150905267,0.988548229,0],[0,0,0,0],[9E+09,9E+09,9E+09,9E+09,9E+09,9E+09]];
  CONST robtarget Target_1650:=[[279.729661692,64.19159225,214.996798109],[0,0.150905267,0.988548229,0],[0,0,0,0],[9E+09,9E+09,9E+09,9E+09,9E+09,9E+09]];
  CONST robtarget Target_1660:=[[280.945624076,64.262977101,214.996798109],[0,0.150905267,0.988548229,0],[0,0,0,0],[9E+09,9E+09,9E+09,9E+09,9E+09,9E+09]];
  CONST robtarget Target_1670:=[[283.732571069,64.043896483,214.996798109],[0,0.150905267,0.988548229,0],[0,0,0,0],[9E+09,9E+09,9E+09,9E+09,9E+09,9E+09]];
  CONST robtarget Target_1680:=[[286.45346803,63.535976952,214.996798109],[0,0.150905267,0.988548229,0],[0,0,0,0],[9E+09,9E+09,9E+09,9E+09,9E+09,9E+09]];
  CONST robtarget Target_1690:=[[288.742098435,62.972912998,214.996798109],[0,0.150905267,0.988548229,0],[0,0,0,0],[9E+09,9E+09,9E+09,9E+09,9E+09,9E+09]];
  CONST robtarget Target_1700:=[[292.303797153,61.991342486,214.996798109],[0,0.150905267,0.988548229,0],[0,0,0,0],[9E+09,9E+09,9E+09,9E+09,9E+09,9E+09]];
  CONST robtarget Target_1710:=[[295.323474875,61.342771747,214.996798109],[0,0.150905267,0.988548229,0],[0,0,0,0],[9E+09,9E+09,9E+09,9E+09,9E+09,9E+09]];
  CONST robtarget Target_1720:=[[298.361489461,60.841502742,214.996798109],[0,0.150905267,0.988548229,0],[0,0,0,0],[9E+09,9E+09,9E+09,9E+09,9E+09,9E+09]];
  CONST robtarget Target_1730:=[[301.381453975,60.587864036,214.996798109],[0,0.150905267,0.988548229,0],[0,0,0,0],[9E+09,9E+09,9E+09,9E+09,9E+09,9E+09]];
  CONST robtarget Target_1740:=[[304.419181769,60.476919409,214.996798109],[0,0.150905267,0.988548229,0],[0,0,0,0],[9E+09,9E+09,9E+09,9E+09,9E+09,9E+09]];
  CONST robtarget Target_1750:=[[305.823944153,60.555611726,214.996798109],[0,0.150905267,0.988548229,0],[0,0,0,0],[9E+09,9E+09,9E+09,9E+09,9E+09,9E+09]];
  CONST robtarget Target_1760:=[[307.839452971,60.804320879,214.996798109],[0,0.150905267,0.988548229,0],[0,0,0,0],[9E+09,9E+09,9E+09,9E+09,9E+09,9E+09]];
  CONST robtarget Target_1770:=[[309.344399588,61.20780969,214.996798109],[0,0.150905267,0.988548229,0],[0,0,0,0],[9E+09,9E+09,9E+09,9E+09,9E+09,9E+09]];
  CONST robtarget Target_1780:=[[310.637356728,61.801774962,214.996798109],[0,0.150905267,0.988548229,0],[0,0,0,0],[9E+09,9E+09,9E+09,9E+09,9E+09,9E+09]];
  CONST robtarget Target_1790:=[[312.391609876,63.105831359,214.996798109],[0,0.150905267,0.988548229,0],[0,0,0,0],[9E+09,9E+09,9E+09,9E+09,9E+09,9E+09]];
  CONST robtarget Target_1800:=[[313.786168948,64.879964281,214.996798109],[0,0.150905267,0.988548229,0],[0,0,0,0],[9E+09,9E+09,9E+09,9E+09,9E+09,9E+09]];
  CONST robtarget Target_1810:=[[314.821293413,66.823617905,214.996798109],[0,0.150905267,0.988548229,0],[0,0,0,0],[9E+09,9E+09,9E+09,9E+09,9E+09,9E+09]];
  CONST robtarget Target_1820:=[[315.519541802,68.424094217,214.996798109],[0,0.150905267,0.988548229,0],[0,0,0,0],[9E+09,9E+09,9E+09,9E+09,9E+09,9E+09]];
  CONST robtarget Target_1830:=[[316.965497265,72.350515519,214.996798109],[0,0.150905267,0.988548229,0],[0,0,0,0],[9E+09,9E+09,9E+09,9E+09,9E+09,9E+09]];
  CONST robtarget Target_1840:=[[318.048989461,75.929643768,214.996798109],[0,0.150905267,0.988548229,0],[0,0,0,0],[9E+09,9E+09,9E+09,9E+09,9E+09,9E+09]];
  CONST robtarget Target_1850:=[[318.806200999,78.649996332,214.996798109],[0,0.150905267,0.988548229,0],[0,0,0,0],[9E+09,9E+09,9E+09,9E+09,9E+09,9E+09]];
  CONST robtarget Target_1860:=[[321.835047153,78.649996332,214.996798109],[0,0.150905267,0.988548229,0],[0,0,0,0],[9E+09,9E+09,9E+09,9E+09,9E+09,9E+09]];
  CONST robtarget Target_1870:=[[321.316970665,76.022937631,214.996798109],[0,0.150905267,0.988548229,0],[0,0,0,0],[9E+09,9E+09,9E+09,9E+09,9E+09,9E+09]];
  CONST robtarget Target_1880:=[[320.931127923,73.673514776,214.996798109],[0,0.150905267,0.988548229,0],[0,0,0,0],[9E+09,9E+09,9E+09,9E+09,9E+09,9E+09]];
  CONST robtarget Target_1890:=[[320.539802408,71.023557328,214.996798109],[0,0.150905267,0.988548229,0],[0,0,0,0],[9E+09,9E+09,9E+09,9E+09,9E+09,9E+09]];
  CONST robtarget Target_1900:=[[320.35022474,68.947563161,214.996798109],[0,0.150905267,0.988548229,0],[0,0,0,0],[9E+09,9E+09,9E+09,9E+09,9E+09,9E+09]];
  CONST robtarget Target_1910:=[[320.389794073,66.260140652,214.996798109],[0,0.150905267,0.988548229,0],[0,0,0,0],[9E+09,9E+09,9E+09,9E+09,9E+09,9E+09]];
  CONST robtarget Target_1920:=[[320.741297153,63.477720691,214.996798109],[0,0.150905267,0.988548229,0],[0,0,0,0],[9E+09,9E+09,9E+09,9E+09,9E+09,9E+09]];
  CONST robtarget Target_1930:=[[321.440572753,60.993804489,214.996798109],[0,0.150905267,0.988548229,0],[0,0,0,0],[9E+09,9E+09,9E+09,9E+09,9E+09,9E+09]];
  CONST robtarget Target_1940:=[[322.479629289,58.791360356,214.996798109],[0,0.150905267,0.988548229,0],[0,0,0,0],[9E+09,9E+09,9E+09,9E+09,9E+09,9E+09]];
  CONST robtarget Target_1950:=[[324.162771512,56.494547614,214.996798109],[0,0.150905267,0.988548229,0],[0,0,0,0],[9E+09,9E+09,9E+09,9E+09,9E+09,9E+09]];
  CONST robtarget Target_1960:=[[325.920129397,54.873411323,214.996798109],[0,0.150905267,0.988548229,0],[0,0,0,0],[9E+09,9E+09,9E+09,9E+09,9E+09,9E+09]];
  CONST robtarget Target_1970:=[[327.691316065,53.736725754,214.996798109],[0,0.150905267,0.988548229,0],[0,0,0,0],[9E+09,9E+09,9E+09,9E+09,9E+09,9E+09]];
  CONST robtarget Target_1980:=[[328.257322794,53.437656588,214.996798109],[0,0.150905267,0.988548229,0],[0,0,0,0],[9E+09,9E+09,9E+09,9E+09,9E+09,9E+09]];
  CONST robtarget Target_1990:=[[331.059639589,52.100628217,214.996798109],[0,0.150905267,0.988548229,0],[0,0,0,0],[9E+09,9E+09,9E+09,9E+09,9E+09,9E+09]];
  CONST robtarget Target_2000:=[[334.988092025,50.380765563,214.996798109],[0,0.150905267,0.988548229,0],[0,0,0,0],[9E+09,9E+09,9E+09,9E+09,9E+09,9E+09]];
  CONST robtarget Target_2010:=[[342.25171382,47.351919409,214.996798109],[0,0.150905267,0.988548229,0],[0,0,0,0],[9E+09,9E+09,9E+09,9E+09,9E+09,9E+09]];
  CONST robtarget Target_2020:=[[344.47889143,46.448622881,214.996798109],[0,0.150905267,0.988548229,0],[0,0,0,0],[9E+09,9E+09,9E+09,9E+09,9E+09,9E+09]];
  CONST robtarget Target_2030:=[[354.533547438,42.425438051,214.996798109],[0,0.150905267,0.988548229,0],[0,0,0,0],[9E+09,9E+09,9E+09,9E+09,9E+09,9E+09]];
  CONST robtarget Target_2040:=[[357.311809974,41.322271973,214.996798109],[0,0.150905267,0.988548229,0],[0,0,0,0],[9E+09,9E+09,9E+09,9E+09,9E+09,9E+09]];
  CONST robtarget Target_2050:=[[363.453636897,38.93845787,214.996798109],[0,0.150905267,0.988548229,0],[0,0,0,0],[9E+09,9E+09,9E+09,9E+09,9E+09,9E+09]];
  CONST robtarget Target_2060:=[[370.156361256,36.330284793,214.996798109],[0,0.150905267,0.988548229,0],[0,0,0,0],[9E+09,9E+09,9E+09,9E+09,9E+09,9E+09]];
  CONST robtarget Target_2070:=[[377.391938179,33.525797614,214.996798109],[0,0.150905267,0.988548229,0],[0,0,0,0],[9E+09,9E+09,9E+09,9E+09,9E+09,9E+09]];
  CONST robtarget Target_2080:=[[385.188412538,30.524996332,214.996798109],[0,0.150905267,0.988548229,0],[0,0,0,0],[9E+09,9E+09,9E+09,9E+09,9E+09,9E+09]];
  CONST robtarget Target_2090:=[[393.545784333,27.327880947,214.996798109],[0,0.150905267,0.988548229,0],[0,0,0,0],[9E+09,9E+09,9E+09,9E+09,9E+09,9E+09]];
  CONST robtarget Target_2100:=[[402.464053564,23.93445146,214.996798109],[0,0.150905267,0.988548229,0],[0,0,0,0],[9E+09,9E+09,9E+09,9E+09,9E+09,9E+09]];
  CONST robtarget Target_2110:=[[411.94322023,20.34470787,214.996798109],[0,0.150905267,0.988548229,0],[0,0,0,0],[9E+09,9E+09,9E+09,9E+09,9E+09,9E+09]];
  CONST robtarget Target_2120:=[[291.041777923,8.229323255,214.996798109],[0,0.707106781,0.707106781,0],[0,0,0,0],[9E+09,9E+09,9E+09,9E+09,9E+09,9E+09]];
  CONST robtarget Target_2130:=[[395.032162538,8.229323255,214.996798109],[0,0.707106781,0.707106781,0],[0,0,0,0],[9E+09,9E+09,9E+09,9E+09,9E+09,9E+09]];
  CONST robtarget Target_2140:=[[404.960047153,8.285412998,214.996798109],[0,0.707106781,0.707106781,0],[0,0,0,0],[9E+09,9E+09,9E+09,9E+09,9E+09,9E+09]];
  CONST robtarget Target_2150:=[[409.545508981,8.344009091,214.996798109],[0,0.707106781,0.707106781,0],[0,0,0,0],[9E+09,9E+09,9E+09,9E+09,9E+09,9E+09]];
  CONST robtarget Target_2160:=[[414.13072023,8.425637357,214.996798109],[0,0.707106781,0.707106781,0],[0,0,0,0],[9E+09,9E+09,9E+09,9E+09,9E+09,9E+09]];
  CONST robtarget Target_2170:=[[418.323974993,8.520502326,214.996798109],[0,0.707106781,0.707106781,0],[0,0,0,0],[9E+09,9E+09,9E+09,9E+09,9E+09,9E+09]];
  CONST robtarget Target_2180:=[[422.516136897,8.649996332,214.996798109],[0,0.707106781,0.707106781,0],[0,0,0,0],[9E+09,9E+09,9E+09,9E+09,9E+09,9E+09]];
  CONST robtarget Target_2190:=[[426.316628484,8.807244007,214.996798109],[0,0.707106781,0.707106781,0],[0,0,0,0],[9E+09,9E+09,9E+09,9E+09,9E+09,9E+09]];
  CONST robtarget Target_2200:=[[430.116297153,8.986534793,214.996798109],[0,0.707106781,0.707106781,0],[0,0,0,0],[9E+09,9E+09,9E+09,9E+09,9E+09,9E+09]];
  CONST robtarget Target_2210:=[[422.544181769,-3.128849822,214.996798109],[0,0.707106781,0.707106781,0],[0,0,0,0],[9E+09,9E+09,9E+09,9E+09,9E+09,9E+09]];
  CONST robtarget Target_2220:=[[422.544181769,-70.520676745,214.996798109],[0,0.707106781,0.707106781,0],[0,0,0,0],[9E+09,9E+09,9E+09,9E+09,9E+09,9E+09]];
  CONST robtarget Target_2230:=[[431.63072023,-79.607215207,214.996798109],[0,0.707106781,0.707106781,0],[0,0,0,0],[9E+09,9E+09,9E+09,9E+09,9E+09,9E+09]];
  CONST robtarget Target_2240:=[[418.000912538,-92.47981136,214.996798109],[0,0.707106781,0.707106781,0],[0,0,0,0],[9E+09,9E+09,9E+09,9E+09,9E+09,9E+09]];
  CONST robtarget Target_2250:=[[418.000912538,-1.614426745,214.996798109],[0,0.707106781,0.707106781,0],[0,0,0,0],[9E+09,9E+09,9E+09,9E+09,9E+09,9E+09]];
  CONST robtarget Target_2260:=[[287.928797153,-1.614426745,214.996798109],[0,0.707106781,0.707106781,0],[0,0,0,0],[9E+09,9E+09,9E+09,9E+09,9E+09,9E+09]];
  CONST robtarget Target_2270:=[[287.928797153,-72.035099822,214.996798109],[0,0.707106781,0.707106781,0],[0,0,0,0],[9E+09,9E+09,9E+09,9E+09,9E+09,9E+09]];
  CONST robtarget Target_2280:=[[297.772547153,-81.878849822,214.996798109],[0,0.707106781,0.707106781,0],[0,0,0,0],[9E+09,9E+09,9E+09,9E+09,9E+09,9E+09]];
  CONST robtarget Target_2290:=[[283.385527923,-95.508657514,214.996798109],[0,0.707106781,0.707106781,0],[0,0,0,0],[9E+09,9E+09,9E+09,9E+09,9E+09,9E+09]];
  CONST robtarget Target_2300:=[[283.385527923,-1.614426745,214.996798109],[0,0.707106781,0.707106781,0],[0,0,0,0],[9E+09,9E+09,9E+09,9E+09,9E+09,9E+09]];
  CONST robtarget Target_2310:=[[275.813412538,5.200477101,214.996798109],[0,0.707106781,0.707106781,0],[0,0,0,0],[9E+09,9E+09,9E+09,9E+09,9E+09,9E+09]];
  CONST robtarget Target_2320:=[[286.442418948,15.044227101,214.996798109],[0,0.707106781,0.707106781,0],[0,0,0,0],[9E+09,9E+09,9E+09,9E+09,9E+09,9E+09]];
  CONST robtarget Target_2330:=[[291.041777923,8.229323255,214.996798109],[0,0.707106781,0.707106781,0],[0,0,0,0],[9E+09,9E+09,9E+09,9E+09,9E+09,9E+09]];
  PROC Path_10()
    MoveL Target_10,v300,fine,MyTool\WObj:=wobj0;
    MoveC Target_20,Target_30,v300,fine,MyTool\WObj:=wobj0;
    MoveC Target_40,Target_50,v300,fine,MyTool\WObj:=wobj0;
    MoveC Target_60,Target_70,v300,fine,MyTool\WObj:=wobj0;
    MoveC Target_80,Target_90,v300,fine,MyTool\WObj:=wobj0;
    MoveL Target_100,v300,fine,MyTool\WObj:=wobj0;
    MoveL Target_110,v300,fine,MyTool\WObj:=wobj0;
    MoveL Target_120,v300,fine,MyTool\WObj:=wobj0;
    MoveC Target_130,Target_140,v300,fine,MyTool\WObj:=wobj0;
    MoveC Target_150,Target_160,v300,fine,MyTool\WObj:=wobj0;
    MoveC Target_170,Target_180,v300,fine,MyTool\WObj:=wobj0;
    MoveC Target_190,Target_200,v300,fine,MyTool\WObj:=wobj0;
    MoveL Target_210,v300,fine,MyTool\WObj:=wobj0;
    MoveC Target_220,Target_230,v300,fine,MyTool\WObj:=wobj0;
    MoveC Target_240,Target_250,v300,fine,MyTool\WObj:=wobj0;
    MoveC Target_260,Target_270,v300,fine,MyTool\WObj:=wobj0;
    MoveC Target_280,Target_290,v300,fine,MyTool\WObj:=wobj0;
    MoveC Target_300,Target_310,v300,fine,MyTool\WObj:=wobj0;
    MoveC Target_320,Target_330,v300,fine,MyTool\WObj:=wobj0;
    MoveC Target_340,Target_350,v300,fine,MyTool\WObj:=wobj0;
    MoveC Target_360,Target_370,v300,fine,MyTool\WObj:=wobj0;
    MoveC Target_380,Target_390,v300,fine,MyTool\WObj:=wobj0;
    MoveC Target_400,Target_410,v300,fine,MyTool\WObj:=wobj0;
    MoveC Target_420,Target_430,v300,fine,MyTool\WObj:=wobj0;
  ENDPROC
  PROC Path_20()
    MoveL Target_440,v300,fine,MyTool\WObj:=wobj0;
    MoveL Target_450,v300,fine,MyTool\WObj:=wobj0;
    MoveL Target_460,v300,fine,MyTool\WObj:=wobj0;
    MoveL Target_470,v300,fine,MyTool\WObj:=wobj0;
    MoveL Target_480,v300,fine,MyTool\WObj:=wobj0;
    MoveL Target_490,v300,fine,MyTool\WObj:=wobj0;
    MoveL Target_500,v300,fine,MyTool\WObj:=wobj0;
    MoveL Target_510,v300,fine,MyTool\WObj:=wobj0;
    MoveL Target_520,v300,fine,MyTool\WObj:=wobj0;
    MoveL Target_530,v300,fine,MyTool\WObj:=wobj0;
    MoveL Target_540,v300,fine,MyTool\WObj:=wobj0;
    MoveL Target_550,v300,fine,MyTool\WObj:=wobj0;
    MoveL Target_560,v300,fine,MyTool\WObj:=wobj0;
    MoveL Target_570,v300,fine,MyTool\WObj:=wobj0;
    MoveL Target_580,v300,fine,MyTool\WObj:=wobj0;
    MoveL Target_590,v300,fine,MyTool\WObj:=wobj0;
    MoveL Target_600,v300,fine,MyTool\WObj:=wobj0;
    MoveL Target_610,v300,fine,MyTool\WObj:=wobj0;
    MoveL Target_620,v300,fine,MyTool\WObj:=wobj0;
    MoveL Target_630,v300,fine,MyTool\WObj:=wobj0;
    MoveL Target_640,v300,fine,MyTool\WObj:=wobj0;
    MoveL Target_650,v300,fine,MyTool\WObj:=wobj0;
    MoveL Target_660,v300,fine,MyTool\WObj:=wobj0;
    MoveL Target_670,v300,fine,MyTool\WObj:=wobj0;
    MoveL Target_680,v300,fine,MyTool\WObj:=wobj0;
    MoveL Target_690,v300,fine,MyTool\WObj:=wobj0;
    MoveL Target_700,v300,fine,MyTool\WObj:=wobj0;
    MoveL Target_710,v300,fine,MyTool\WObj:=wobj0;
    MoveL Target_720,v300,fine,MyTool\WObj:=wobj0;
    MoveL Target_730,v300,fine,MyTool\WObj:=wobj0;
    MoveL Target_740,v300,fine,MyTool\WObj:=wobj0;
    MoveL Target_750,v300,fine,MyTool\WObj:=wobj0;
    MoveL Target_760,v300,fine,MyTool\WObj:=wobj0;
    MoveL Target_770,v300,fine,MyTool\WObj:=wobj0;
    MoveL Target_780,v300,fine,MyTool\WObj:=wobj0;
    MoveL Target_790,v300,fine,MyTool\WObj:=wobj0;
    MoveL Target_800,v300,fine,MyTool\WObj:=wobj0;
    MoveL Target_810,v300,fine,MyTool\WObj:=wobj0;
    MoveL Target_820,v300,fine,MyTool\WObj:=wobj0;
    MoveL Target_830,v300,fine,MyTool\WObj:=wobj0;
    MoveL Target_840,v300,fine,MyTool\WObj:=wobj0;
    MoveL Target_850,v300,fine,MyTool\WObj:=wobj0;
    MoveL Target_860,v300,fine,MyTool\WObj:=wobj0;
    MoveL Target_870,v300,fine,MyTool\WObj:=wobj0;
    MoveL Target_880,v300,fine,MyTool\WObj:=wobj0;
    MoveL Target_890,v300,fine,MyTool\WObj:=wobj0;
    MoveL Target_900,v300,fine,MyTool\WObj:=wobj0;
    MoveL Target_910,v300,fine,MyTool\WObj:=wobj0;
    MoveL Target_920,v300,fine,MyTool\WObj:=wobj0;
    MoveL Target_930,v300,fine,MyTool\WObj:=wobj0;
    MoveL Target_940,v300,fine,MyTool\WObj:=wobj0;
    MoveL Target_950,v300,fine,MyTool\WObj:=wobj0;
    MoveL Target_960,v300,fine,MyTool\WObj:=wobj0;
    MoveL Target_970,v300,fine,MyTool\WObj:=wobj0;
    MoveL Target_980,v300,fine,MyTool\WObj:=wobj0;
    MoveL Target_990,v300,fine,MyTool\WObj:=wobj0;
    MoveL Target_1000,v300,fine,MyTool\WObj:=wobj0;
    MoveL Target_1010,v300,fine,MyTool\WObj:=wobj0;
    MoveL Target_1020,v300,fine,MyTool\WObj:=wobj0;
    MoveL Target_1030,v300,fine,MyTool\WObj:=wobj0;
    MoveL Target_1040,v300,fine,MyTool\WObj:=wobj0;
    MoveL Target_1050,v300,fine,MyTool\WObj:=wobj0;
    MoveL Target_1060,v300,fine,MyTool\WObj:=wobj0;
    MoveL Target_1070,v300,fine,MyTool\WObj:=wobj0;
    MoveL Target_1080,v300,fine,MyTool\WObj:=wobj0;
    MoveL Target_1090,v300,fine,MyTool\WObj:=wobj0;
    MoveL Target_1100,v300,fine,MyTool\WObj:=wobj0;
    MoveL Target_1110,v300,fine,MyTool\WObj:=wobj0;
    MoveL Target_1120,v300,fine,MyTool\WObj:=wobj0;
    MoveL Target_1130,v300,fine,MyTool\WObj:=wobj0;
    MoveL Target_1140,v300,fine,MyTool\WObj:=wobj0;
    MoveL Target_1150,v300,fine,MyTool\WObj:=wobj0;
    MoveL Target_1160,v300,fine,MyTool\WObj:=wobj0;
    MoveL Target_1170,v300,fine,MyTool\WObj:=wobj0;
    MoveL Target_1180,v300,fine,MyTool\WObj:=wobj0;
    MoveL Target_1190,v300,fine,MyTool\WObj:=wobj0;
    MoveL Target_1200,v300,fine,MyTool\WObj:=wobj0;
    MoveL Target_1210,v300,fine,MyTool\WObj:=wobj0;
    MoveL Target_1220,v300,fine,MyTool\WObj:=wobj0;
    MoveL Target_1230,v300,fine,MyTool\WObj:=wobj0;
    MoveL Target_1240,v300,fine,MyTool\WObj:=wobj0;
    MoveL Target_1250,v300,fine,MyTool\WObj:=wobj0;
    MoveL Target_1260,v300,fine,MyTool\WObj:=wobj0;
  ENDPROC
  PROC Path_30()
    MoveL Target_1270,v300,fine,MyTool\WObj:=wobj0;
    MoveL Target_1280,v300,fine,MyTool\WObj:=wobj0;
    MoveL Target_1290,v300,fine,MyTool\WObj:=wobj0;
    MoveL Target_1300,v300,fine,MyTool\WObj:=wobj0;
    MoveL Target_1310,v300,fine,MyTool\WObj:=wobj0;
    MoveL Target_1320,v300,fine,MyTool\WObj:=wobj0;
    MoveL Target_1330,v300,fine,MyTool\WObj:=wobj0;
    MoveL Target_1340,v300,fine,MyTool\WObj:=wobj0;
    MoveL Target_1350,v300,fine,MyTool\WObj:=wobj0;
    MoveL Target_1360,v300,fine,MyTool\WObj:=wobj0;
    MoveL Target_1370,v300,fine,MyTool\WObj:=wobj0;
    MoveL Target_1380,v300,fine,MyTool\WObj:=wobj0;
    MoveC Target_1390,Target_1400,v300,fine,MyTool\WObj:=wobj0;
    MoveC Target_1410,Target_1420,v300,fine,MyTool\WObj:=wobj0;
    MoveL Target_1430,v300,fine,MyTool\WObj:=wobj0;
    MoveL Target_1440,v300,fine,MyTool\WObj:=wobj0;
    MoveL Target_1450,v300,fine,MyTool\WObj:=wobj0;
    MoveL Target_1460,v300,fine,MyTool\WObj:=wobj0;
    MoveL Target_1470,v300,fine,MyTool\WObj:=wobj0;
    MoveL Target_1480,v300,fine,MyTool\WObj:=wobj0;
    MoveC Target_1490,Target_1500,v300,fine,MyTool\WObj:=wobj0;
    MoveC Target_1510,Target_1520,v300,fine,MyTool\WObj:=wobj0;
    MoveC Target_1530,Target_1540,v300,fine,MyTool\WObj:=wobj0;
    MoveC Target_1550,Target_1560,v300,fine,MyTool\WObj:=wobj0;
    MoveC Target_1570,Target_1580,v300,fine,MyTool\WObj:=wobj0;
    MoveC Target_1590,Target_1600,v300,fine,MyTool\WObj:=wobj0;
    MoveC Target_1610,Target_1620,v300,fine,MyTool\WObj:=wobj0;
    MoveC Target_1630,Target_1640,v300,fine,MyTool\WObj:=wobj0;
    MoveC Target_1650,Target_1660,v300,fine,MyTool\WObj:=wobj0;
    MoveC Target_1670,Target_1680,v300,fine,MyTool\WObj:=wobj0;
    MoveC Target_1690,Target_1700,v300,fine,MyTool\WObj:=wobj0;
    MoveC Target_1710,Target_1720,v300,fine,MyTool\WObj:=wobj0;
    MoveC Target_1730,Target_1740,v300,fine,MyTool\WObj:=wobj0;
    MoveC Target_1750,Target_1760,v300,fine,MyTool\WObj:=wobj0;
    MoveC Target_1770,Target_1780,v300,fine,MyTool\WObj:=wobj0;
    MoveC Target_1790,Target_1800,v300,fine,MyTool\WObj:=wobj0;
    MoveC Target_1810,Target_1820,v300,fine,MyTool\WObj:=wobj0;
    MoveC Target_1830,Target_1840,v300,fine,MyTool\WObj:=wobj0;
    MoveL Target_1850,v300,fine,MyTool\WObj:=wobj0;
    MoveL Target_1860,v300,fine,MyTool\WObj:=wobj0;
    MoveC Target_1870,Target_1880,v300,fine,MyTool\WObj:=wobj0;
    MoveL Target_1890,v300,fine,MyTool\WObj:=wobj0;
    MoveC Target_1900,Target_1910,v300,fine,MyTool\WObj:=wobj0;
    MoveC Target_1920,Target_1930,v300,fine,MyTool\WObj:=wobj0;
    MoveC Target_1940,Target_1950,v300,fine,MyTool\WObj:=wobj0;
    MoveC Target_1960,Target_1970,v300,fine,MyTool\WObj:=wobj0;
    MoveL Target_1980,v300,fine,MyTool\WObj:=wobj0;
    MoveC Target_1990,Target_2000,v300,fine,MyTool\WObj:=wobj0;
    MoveL Target_2010,v300,fine,MyTool\WObj:=wobj0;
    MoveL Target_2020,v300,fine,MyTool\WObj:=wobj0;
    MoveL Target_2030,v300,fine,MyTool\WObj:=wobj0;
    MoveL Target_2040,v300,fine,MyTool\WObj:=wobj0;
    MoveL Target_2050,v300,fine,MyTool\WObj:=wobj0;
    MoveL Target_2060,v300,fine,MyTool\WObj:=wobj0;
    MoveL Target_2070,v300,fine,MyTool\WObj:=wobj0;
    MoveL Target_2080,v300,fine,MyTool\WObj:=wobj0;
    MoveL Target_2090,v300,fine,MyTool\WObj:=wobj0;
    MoveL Target_2100,v300,fine,MyTool\WObj:=wobj0;
    MoveL Target_2110,v300,fine,MyTool\WObj:=wobj0;
  ENDPROC
  PROC Path_40()
    MoveL Target_2120,v300,fine,MyTool\WObj:=wobj0;
    MoveL Target_2130,v300,fine,MyTool\WObj:=wobj0;
    MoveL Target_2140,v300,fine,MyTool\WObj:=wobj0;
    MoveL Target_2150,v300,fine,MyTool\WObj:=wobj0;
    MoveL Target_2160,v300,fine,MyTool\WObj:=wobj0;
    MoveL Target_2170,v300,fine,MyTool\WObj:=wobj0;
    MoveL Target_2180,v300,fine,MyTool\WObj:=wobj0;
    MoveL Target_2190,v300,fine,MyTool\WObj:=wobj0;
    MoveL Target_2200,v300,fine,MyTool\WObj:=wobj0;
    MoveL Target_2210,v300,fine,MyTool\WObj:=wobj0;
    MoveL Target_2220,v300,fine,MyTool\WObj:=wobj0;
    MoveL Target_2230,v300,fine,MyTool\WObj:=wobj0;
    MoveL Target_2240,v300,fine,MyTool\WObj:=wobj0;
    MoveL Target_2250,v300,fine,MyTool\WObj:=wobj0;
    MoveL Target_2260,v300,fine,MyTool\WObj:=wobj0;
    MoveL Target_2270,v300,fine,MyTool\WObj:=wobj0;
    MoveL Target_2280,v300,fine,MyTool\WObj:=wobj0;
    MoveL Target_2290,v300,fine,MyTool\WObj:=wobj0;
    MoveL Target_2300,v300,fine,MyTool\WObj:=wobj0;
    MoveL Target_2310,v300,fine,MyTool\WObj:=wobj0;
    MoveL Target_2320,v300,fine,MyTool\WObj:=wobj0;
    MoveL Target_2330,v300,fine,MyTool\WObj:=wobj0;
  ENDPROC
ENDMODULE

